(* IEC 61131-3 sources: Industry-PLC-LLM/data/PLCBEAD_repo/PLCBEAD_PLCEmbed-main/PLC-BEAD/Source/GEB/HOLIDAY, 1 file *)

(* ---- HOLIDAY.ST ---- *)
TYPE oscat_LANGUAGE:
  STRUCT
    DEFAULT 	: INT;
	LMAX    	: INT;
  END_STRUCT;
END_TYPE

TYPE
	oscat_LOCATION_ELEMENTS	: ARRAY [1..5] OF INT;
END_TYPE

TYPE
  oscat_ELEMENT_WEEKDAYS	: ARRAY [1..7] OF STRING;
  oscat_WEEKDAYS			: ARRAY [1..3]  OF oscat_ELEMENT_WEEKDAYS;
END_TYPE

TYPE oscat_LOCATION:
  STRUCT
    DEFAULT 	: INT;
	LMAX    	: INT;
	LANGUAGE	: oscat_LOCATION_ELEMENTS;
  END_STRUCT;
END_TYPE

TYPE oscat_HOLIDAY_DATA :
  STRUCT
	NAME : STRING;
	DAY  : SINT;
	MONTH : SINT;
	USE : SINT;
	PAD_BYTE : BYTE;
  END_STRUCT;
END_TYPE

TYPE
  oscat_HOLIDAY_DATA_0_29 	: ARRAY [0..29] OF oscat_HOLIDAY_DATA;
  oscat_HOLIDAY_DATA_0_49 	: ARRAY [0..49] OF oscat_HOLIDAY_DATA;
END_TYPE

FUNCTION_BLOCK SETUP_LANGUAGE_Block

	VAR_IN_OUT
		LANGUAGE :	oscat_LANGUAGE;
	END_VAR

	VAR
		init :	BOOL;
	END_VAR

	IF init THEN RETURN; END_IF;
	init := TRUE;

	LANGUAGE.DEFAULT  := 1; (* 1=english, 2=german 3=french *)
	LANGUAGE.LMAX := 3;
END_FUNCTION_BLOCK

FUNCTION_BLOCK SETUP_LOCATION
	VAR_IN_OUT
		LOCATION :	oscat_LOCATION;
	END_VAR

	VAR
		init :	BOOL;
	END_VAR

	IF init THEN RETURN; END_IF;
	init := TRUE;

	LOCATION.DEFAULT  := 1;
	LOCATION.LMAX := 5;

	LOCATION.LANGUAGE[1] := 2;
	LOCATION.LANGUAGE[2] := 2;
	LOCATION.LANGUAGE[3] := 3;
	LOCATION.LANGUAGE[4] := 2;
	LOCATION.LANGUAGE[5] := 2;
END_FUNCTION_BLOCK

FUNCTION_BLOCK SETUP_WEEKDAYS

	VAR_IN_OUT
		WEEKDAYS :	oscat_WEEKDAYS;
	END_VAR

	VAR
		init :	BOOL;
	END_VAR

	IF init THEN RETURN; END_IF;
	init := TRUE;

	WEEKDAYS[1][01] := 'MonDAY';
	WEEKDAYS[1][02] := 'TuesDAY';
	WEEKDAYS[1][03] := 'WednesDAY';
	WEEKDAYS[1][04] := 'ThursDAY';
	WEEKDAYS[1][05] := 'FriDAY';
	WEEKDAYS[1][06] := 'SaturDAY';
	WEEKDAYS[1][07] := 'SunDAY';

	WEEKDAYS[2][01] := 'Montag';
	WEEKDAYS[2][02] := 'Dienstag';
	WEEKDAYS[2][03] := 'Mittwoch';
	WEEKDAYS[2][04] := 'Donnerstag';
	WEEKDAYS[2][05] := 'Freitag';
	WEEKDAYS[2][06] := 'Samstag';
	WEEKDAYS[2][07] := 'Sonntag';

	WEEKDAYS[3][01] := 'Lundi';
	WEEKDAYS[3][02] := 'Mardi';
	WEEKDAYS[3][03] := 'Mercredi';
	WEEKDAYS[3][04] := 'Jeudi';
	WEEKDAYS[3][05] := 'Vendredi';
	WEEKDAYS[3][06] := 'Samedi';
	WEEKDAYS[3][07] := 'Dimanche';
END_FUNCTION_BLOCK

FUNCTION YEAR_OF_DATE:INT
	VAR_INPUT
		IDATE :	UDINT;
	END_VAR

	YEAR_OF_DATE := UDINT_TO_INT((IDATE+UDINT#43200) / UDINT#31557600 + UDINT#1970);
END_FUNCTION

FUNCTION _INT_TO_UDINT:UDINT
	VAR_INPUT
		IN :	INT;
	END_VAR

	_INT_TO_UDINT := DINT_TO_UDINT(INT_TO_DINT(IN));
END_FUNCTION

FUNCTION SET_DATE:UDINT

	VAR_INPUT
		YEAR  :	INT;
		MONTH :	INT;
		DAY  :	INT;
	END_VAR

	VAR
		count :	INT;
	END_VAR

	IF MONTH > 2 THEN
		count := (MONTH - 1) * 30;
		IF MONTH > 7 THEN
			count := count + DWORD_TO_INT(SHR(DINT_TO_DWORD(INT_TO_DINT(MONTH) - INT_TO_DINT(3)),1));
		ELSE
			count := count + DWORD_TO_INT(SHR(DINT_TO_DWORD(INT_TO_DINT(MONTH) - INT_TO_DINT(4)),1));
		END_IF;
		IF SHL(INT_TO_WORD(YEAR),14) = WORD#0 THEN
			count := count + 1;
		END_IF;
	ELSE
		count := (MONTH - 1) * 31;
	END_IF;
	SET_DATE := (_INT_TO_UDINT(count + DAY  - 1) + DWORD_TO_UDINT(SHR(UDINT_TO_DWORD(_INT_TO_UDINT(YEAR) * UDINT#1461 - UDINT#2878169), 2))) * UDINT#86400;
END_FUNCTION

FUNCTION DAY_OF_WEEK:INT
	VAR_INPUT
		IDATE :	UDINT;
	END_VAR

	DAY_OF_WEEK := UDINT_TO_INT((IDATE / UDINT#86400 + UDINT#3) MOD UDINT#7) + INT#01;
END_FUNCTION

FUNCTION EASTER:UDINT
	VAR_INPUT
		YEAR  :	INT;
	END_VAR

	VAR
		b :	INT;
		c :	INT;
		oDAY  :	INT;
	END_VAR

	b := (204 - 11 * (YEAR  MOD 19)) MOD 30;
	IF b > 27 THEN b := b - 1; END_IF;
	c := (YEAR  + WORD_TO_INT(SHR(INT_TO_WORD(YEAR),2)) + b - 13) MOD 7;
	oDAY  := 28 + b - c;
	IF oDAY  > 33 THEN
		EASTER := SET_DATE(YEAR, 4, oDAY  - 31);
	ELSE
		EASTER := SET_DATE(YEAR, 3, oDAY);
	END_IF;
END_FUNCTION

FUNCTION LEAP_OF_DATE:BOOL

	VAR_INPUT
		IDATE :	UDINT;
	END_VAR

	LEAP_OF_DATE := SHL(UDINT_TO_DWORD((IDATE + UDINT#43200) / UDINT#31557600), 30) = DWORD#16#80000000;
END_FUNCTION

FUNCTION DAY_OF_YEAR:INT
	VAR_INPUT
		IDATE :	UDINT;
	END_VAR

	DAY_OF_YEAR  := UDINT_TO_INT(((IDATE) / UDINT#86400) MOD UDINT#1461);
	IF DAY_OF_YEAR  > 729 THEN
		IF DAY_OF_YEAR  > 1095 THEN DAY_OF_YEAR  := DAY_OF_YEAR  - 1095; ELSE DAY_OF_YEAR  := DAY_OF_YEAR  - 729; END_IF;
	ELSIF DAY_OF_YEAR  > 364 THEN
		DAY_OF_YEAR  := DAY_OF_YEAR  - 364;
	ELSE
		DAY_OF_YEAR  := DAY_OF_YEAR  + 1;
	END_IF;
END_FUNCTION

FUNCTION MONTH_OF_DATE:INT

	VAR_INPUT
		IDATE :	UDINT;
	END_VAR

	MONTH_OF_DATE := DAY_OF_YEAR(IDATE);
	IF MONTH_OF_DATE < 32 THEN
		MONTH_OF_DATE := 1;
	ELSIF LEAP_OF_DATE((IDATE)) THEN
		MONTH_OF_DATE := (MONTH_OF_DATE * 53 + 1668) / 1623;
	ELSE
		MONTH_OF_DATE := (MONTH_OF_DATE * 53 + 1700) / 1620;
	END_IF;
END_FUNCTION

FUNCTION DAY_OF_MONTH:INT
	VAR_INPUT
		IDATE :	UDINT;
	END_VAR

	DAY_OF_MONTH := DAY_OF_YEAR(IDATE);

	IF LEAP_OF_DATE((IDATE)) THEN
		CASE DAY_OF_MONTH OF
			32..60	:	DAY_OF_MONTH := DAY_OF_MONTH - 31;
			61..91	:	DAY_OF_MONTH := DAY_OF_MONTH - 60;
			92..121 :	DAY_OF_MONTH := DAY_OF_MONTH - 91;
			122..152:	DAY_OF_MONTH := DAY_OF_MONTH - 121;
			153..182:	DAY_OF_MONTH := DAY_OF_MONTH - 152;
			183..213:	DAY_OF_MONTH := DAY_OF_MONTH - 182;
			214..244:	DAY_OF_MONTH := DAY_OF_MONTH - 213;
			245..274:	DAY_OF_MONTH := DAY_OF_MONTH - 244;
			275..305:	DAY_OF_MONTH := DAY_OF_MONTH - 274;
			306..335:	DAY_OF_MONTH := DAY_OF_MONTH - 305;
			336..366:	DAY_OF_MONTH := DAY_OF_MONTH - 335;
		END_CASE;
	ELSE
		CASE DAY_OF_MONTH OF
			32..59	:	DAY_OF_MONTH := DAY_OF_MONTH - 31;
			60..90	:	DAY_OF_MONTH := DAY_OF_MONTH - 59;
			91..120 :	DAY_OF_MONTH := DAY_OF_MONTH - 90;
			121..151:	DAY_OF_MONTH := DAY_OF_MONTH - 120;
			152..181:	DAY_OF_MONTH := DAY_OF_MONTH - 151;
			182..212:	DAY_OF_MONTH := DAY_OF_MONTH - 181;
			213..243:	DAY_OF_MONTH := DAY_OF_MONTH - 212;
			244..273:	DAY_OF_MONTH := DAY_OF_MONTH - 243;
			274..304:	DAY_OF_MONTH := DAY_OF_MONTH - 273;
			305..334:	DAY_OF_MONTH := DAY_OF_MONTH - 304;
			335..365:	DAY_OF_MONTH := DAY_OF_MONTH - 334;
		END_CASE;
	END_IF;
END_FUNCTION

FUNCTION DATE_ADD:UDINT
	VAR_INPUT
		IDATE :	UDINT;
		D :	INT;
		W :	INT;
		M :	INT;
		Y :	INT;
	END_VAR

	VAR
		mo :	INT;
		yr :	INT;
		dm :	INT;
	END_VAR

	DATE_ADD := IDATE + INT_TO_UDINT(D + W * 7) * UDINT#86400;
	yr := Y + YEAR_OF_DATE(DATE_ADD);
	mo := M + MONTH_OF_DATE(DATE_ADD);
	dm := DAY_OF_MONTH(DATE_ADD);
	WHILE mo > 12 DO
		mo := mo - 12;
		yr := yr + 1;
	END_WHILE;
	WHILE mo < 1 DO
		mo := mo + 12;
		yr := yr - 1;
	END_WHILE;
	DATE_ADD := SET_DATE(yr, mo, dm);
END_FUNCTION

FUNCTION_BLOCK HOLIDAY_Block
	VAR_INPUT
		DATE_IN :	UDINT;
		LANGU :	INT;
		FRIDAY  :	BOOL;
		SATURDAY  :	BOOL;
		SUNDAY  :	BOOL;
	END_VAR

	VAR_IN_OUT
		HOLIDAYS :	oscat_HOLIDAY_DATA_0_29;
	END_VAR

	VAR_OUTPUT
		Y :	BOOL;
		NAME :	STRING;
	END_VAR

	VAR
		SIZE :	INT := INT#29;
		last_active :	UDINT;
		ostern :	UDINT;
		i :	INT;
		jahr :	INT;
		x_date :	UDINT;
		lx :	INT;
		wdx :	INT;
		SETUP_LOCATIONS :	SETUP_LOCATION;
		SETUP_WEEKDAYSS :	SETUP_WEEKDAYS;
		SETUP_LANGUAGES :	SETUP_LANGUAGE_Block;
		LOCATION :	oscat_LOCATION;
		WEEKDAYS :	oscat_WEEKDAYS;
		LANGUAGE :	oscat_LANGUAGE;
		wd :	INT;
	END_VAR

	IF last_active = DATE_IN THEN RETURN; END_IF;
	last_active := DATE_IN;

	SETUP_LOCATIONS(LOCATION:=LOCATION);
	LOCATION:=SETUP_LOCATIONS.LOCATION;

	SETUP_WEEKDAYSS(WEEKDAYS:=WEEKDAYS);
	WEEKDAYS:=SETUP_WEEKDAYSS.WEEKDAYS;

	SETUP_LANGUAGES(LANGUAGE:=LANGUAGE);
	LANGUAGE:=SETUP_LANGUAGES.LANGUAGE;

	IF LANGU = 0 THEN
		lx := LANGUAGE.DEFAULT;
	ELSE
		lx := MIN(LANGUAGE.LMAX, LANGU);
	END_IF;

	jahr := YEAR_OF_DATE(DATE_IN);
	ostern := EASTER(jahr);
	wdx := DAY_OF_WEEK(DATE_IN);
	Y := FALSE;

	FOR i := 0 TO SIZE DO
		x_date := SET_DATE(jahr, SINT_TO_INT(HOLIDAYS[i].MONTH) , SINT_TO_INT(HOLIDAYS[i].DAY));
		IF HOLIDAYS[i].USE = SINT#1 AND HOLIDAYS[i].MONTH > SINT#0 THEN
			(* check for fixed date holiDAY  *)
			IF x_date = DATE_IN THEN
				Y := TRUE;
				NAME := HOLIDAYS[i].NAME;
				RETURN;
			END_IF;
		ELSIF HOLIDAYS[i].USE = SINT#1 AND HOLIDAYS[i].MONTH = SINT#0 THEN
			(* check for holiDAY  IN reference to EASTER *)
			IF DATE_ADD(ostern, SINT_TO_INT(HOLIDAYS[i].DAY),0,0,0) = DATE_IN THEN
				Y := TRUE;
				NAME := HOLIDAYS[i].NAME;
				RETURN;
			END_IF;
		ELSIF HOLIDAYS[i].USE < SINT#0 THEN
			(* check for holiDAY  on a weekDAY  before date *)
			IF DAY_OF_WEEK(DATE_IN) = SINT_TO_INT(ABS(HOLIDAYS[i].USE)) AND DATE_IN < x_date AND DATE_IN >= DATE_ADD(x_date,-7,0,0,0) THEN
				Y := TRUE;
				NAME := HOLIDAYS[i].NAME;
				RETURN;
			END_IF;
		END_IF;
	END_FOR;

	IF NOT Y AND (wdx = 5 AND FRIDAY  OR wdx = 6 AND SATURDAY  OR wdx = 7 AND SUNDAY) THEN
		Y := TRUE;
		wd := LOCATION.LANGUAGE[lx];
		NAME := WEEKDAYS[wd][wdx];
	ELSE
		NAME := '';
	END_IF;
END_FUNCTION_BLOCK

PROGRAM program0
  VAR
	DATE_IN  :	UDINT;
	LANGU    :	INT;
	FRIDAY    :	BOOL;
	SATURDAY  :	BOOL;
	SUNDAY    :	BOOL;

	Y :	BOOL;
	NAME :	STRING;

	HOLIDAYS :	oscat_HOLIDAY_DATA_0_29;

	func_block : HOLIDAY_Block;
  END_VAR
	func_block.DATE_IN :=DATE_IN ;
	func_block.LANGU   :=LANGU   ;
	func_block.FRIDAY   :=FRIDAY   ;
	func_block.SATURDAY:=SATURDAY;
	func_block.SUNDAY   :=SUNDAY   ;

	func_block(HOLIDAYS  :=HOLIDAYS );
	Y := func_block.Y;
	NAME := func_block.NAME;
	HOLIDAYS := func_block.HOLIDAYS;

END_PROGRAM
